(* PLC project test1.project, CODESYS CODESYS V3.5 SP14 *)
(* stored: creationDateTime 2019-01-04T21:29:38.833276, modificationDateTime 2019-01-04T21:22:27.3042161 *)

PROGRAM PLC_PRG
  VAR
    Start_PB : BOOL;  (* スタートボタン *)
    Start_PB_push : BOOL;  (* スタートボタンが押された自己保持 *)
    Lamp : BOOL;  (* ランプ点灯！ *)
    elapsed_time_on : TIME;  (* 実際の点灯時間 *)
    Lamp_off : BOOL;  (* ランプ消灯命令 *)
    off_interval_time : TIME := TIME#1s0ms;  (* ランプ消灯時間設定値[ms] *)
    elapsed_time_off : TIME;  (* ランプ消灯時間実測値[ms] *)
    Lamp_off_interval_timer : TON;  (* ランプ消灯時間設定タイマー *)
    Lamp_on_interval_timer : TON;  (* ランプ点灯時間設定タイマー *)
    on_interval_time : TIME := TIME#2s0ms;  (* ランプ点灯時間設定値 *)
    Stop_PB : BOOL;  (* 停止ボタン *)
    go : BOOL;
  END_VAR

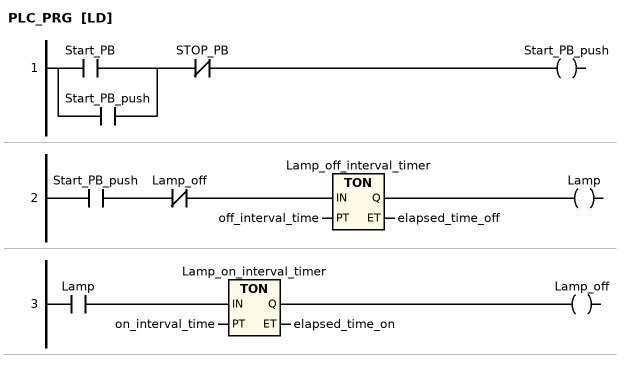
(* LD diagram, written out as Structured Text *)

Start_PB_push := (Start_PB OR Start_PB_push) AND NOT STOP_PB;

Lamp_off_interval_timer(IN := Start_PB_push AND NOT Lamp_off, PT := off_interval_time, ET => elapsed_time_off);
Lamp := Lamp_off_interval_timer.Q;

Lamp_on_interval_timer(IN := Lamp, PT := on_interval_time, ET => elapsed_time_on);
Lamp_off := Lamp_on_interval_timer.Q;
END_PROGRAM
